FUNCTION_BLOCK PUBLIC FB_MyOpcUaMethod
VAR_INPUT
	in1 : INT;
	in2 : INT;
END_VAR
VAR_OUTPUT
	result : INT;
END_VAR

{attribute 'TcRpcEnable' := '1'}
METHOD PUBLIC Multiply : INT
VAR_INPUT
	a : INT;
	b : INT;
END_VAR
Multiply := a * b;
END_METHOD

END_FUNCTION_BLOCK

(* stored: Version 1.1.0.1, ProductVersion 3.1.4026.18
   POU FB_MyOpcUaMethod: Id {fd6aedc3-3cae-4807-bc00-d82107da6d27}, SpecialFunc None
   Method Multiply: Id {bacdc101-7811-4568-b8f7-d894b6cac98a} *)
